{attribute 'qualified_only'}
{attribute 'strict'}
TYPE EAbortState :
(
	none := 0,
	requested := 1,
	aborting := 2,
	aborted := 3
);
END_TYPE

(* stored: Version 1.1.0.1
   DUT EAbortState: Id {fa221045-acf4-4ffc-9a76-99606418d2e2} *)
